Fanuc KAREL source: kb00197.KL

-- PROVISIONAL review KL for V1013-1; original PC SHA256 a99e797f25c74c790466f9238d1d8e605ea87a6835171cc60c7cf56805593a3f
-- Incomplete behavior may be omitted. Consult companion uncertainty JSON. Do not deploy.
PROGRAM KB00197
%NOLOCKGROUP
BEGIN
  -- UNRESOLVED_PC offsets 5-14; opcodes 3F,75
  -- UNRESOLVED_PC offsets 19-26; opcodes 9D,23
  -- UNRESOLVED_PC offsets 31-38; opcodes 9D,23
  -- UNRESOLVED_PC offsets 43-73; opcodes 27,22,22,2A,22,22,31
  -- UNRESOLVED_PC offsets 78-82; opcodes 7F
END KB00197
